// TIA Portal V20 export
// export: Created 2025-12-01T14:56:18.0227958Z, ExportSetting None, DisplayName Totally Integrated Automation Portal, DisplayVersion V20 Update 3, DisplayName TIA Portal Openness, DisplayVersion V20 Update 3, DisplayName TIA Portal Version Control Interface, DisplayVersion V20 Update 3, DisplayName STEP 7 Professional, DisplayVersion V20 Update 3, DisplayName STEP 7 Safety, DisplayVersion V20 Update 2, DisplayName WinCC Basic/Comfort/Advanced, DisplayVersion V20 Update 3, DisplayName WinCC Professional, DisplayVersion V20 Update 3, DisplayName WinCC Unified, DisplayVersion V20 Update 3
TYPE "UDT_HMI_SeñalesBarreras"
   STRUCT
      MS_11 : Bool;
      MS_12 : Bool;
      MS_21 : Bool;
      MS_22 : Bool;
      STOP : Bool;
      FREE : Bool;
      ENABLE : Bool;
      ACK : Bool;
      Q : Bool;
      MUTING : Bool;
      ACK_REQ : Bool;
      FAULT : Bool;
      Reserva_14 : Bool;
      Reserva_15 : Bool;
      Reserva_16 : Bool;
      Reserva_17 : Bool;
   END_STRUCT;
END_TYPE
